ABB RAPID module: Module1.mod

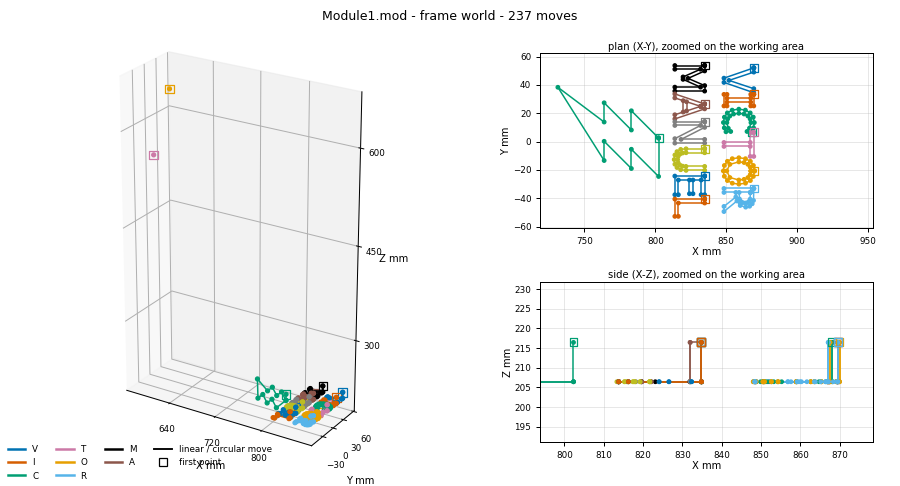
[picture p0: tool path of Module1.mod in frame world, 237 of 237 moves have a stored position in this frame; points joined in program order, loops and branches not executed]
MODULE Module1
        CONST robtarget Target_10_2:=[[151.956,135.501,-10],[0.707106781,0,0,0.707106781],[0,-2,1,0],[9E+09,9E+09,9E+09,9E+09,9E+09,9E+09]];
    CONST robtarget Target_10:=[[151.956,135.501,0],[0.707106781,0,0,0.707106781],[0,0,0,0],[9E+09,9E+09,9E+09,9E+09,9E+09,9E+09]];
    CONST robtarget Target_20:=[[154.96,135.501,0],[0.707106781,0,0,0.707106781],[0,-2,1,0],[9E+09,9E+09,9E+09,9E+09,9E+09,9E+09]];
    CONST robtarget Target_30:=[[160.796,152.992,0],[0.707106781,0,0,0.707106781],[0,-2,1,0],[9E+09,9E+09,9E+09,9E+09,9E+09,9E+09]];
    CONST robtarget Target_40:=[[166.632,135.501,0],[0.707106781,0,0,0.707106781],[0,-2,1,0],[9E+09,9E+09,9E+09,9E+09,9E+09,9E+09]];
    CONST robtarget Target_50:=[[169.481,135.501,0],[0.707106781,0,0,0.707106781],[0,-2,1,0],[9E+09,9E+09,9E+09,9E+09,9E+09,9E+09]];
    CONST robtarget Target_60:=[[162.229,156.559,0],[0.707106781,0,0,0.707106781],[0,-2,1,0],[9E+09,9E+09,9E+09,9E+09,9E+09,9E+09]];
    CONST robtarget Target_70:=[[159.209,156.559,0],[0.707106781,0,0,0.707106781],[0,-2,1,0],[9E+09,9E+09,9E+09,9E+09,9E+09,9E+09]];
    CONST robtarget Target_80:=[[151.956,135.501,0],[0.707106781,0,0,0.707106781],[0,-2,1,0],[9E+09,9E+09,9E+09,9E+09,9E+09,9E+09]];
    CONST robtarget Target_90_2:=[[170.676,135.501,-10],[0.707106781,0,0,0.707106781],[0,-2,1,0],[9E+09,9E+09,9E+09,9E+09,9E+09,9E+09]];
    CONST robtarget Target_90:=[[170.676,135.501,0],[0.707106781,0,0,0.707106781],[0,-2,1,0],[9E+09,9E+09,9E+09,9E+09,9E+09,9E+09]];
    CONST robtarget Target_100:=[[178.833,135.501,0],[0.707106781,0,0,0.707106781],[0,-2,1,0],[9E+09,9E+09,9E+09,9E+09,9E+09,9E+09]];
    CONST robtarget Target_110:=[[178.833,137.651,0],[0.707106781,0,0,0.707106781],[0,-2,1,0],[9E+09,9E+09,9E+09,9E+09,9E+09,9E+09]];
    CONST robtarget Target_120:=[[176.153,137.651,0],[0.707106781,0,0,0.707106781],[0,-2,1,0],[9E+09,9E+09,9E+09,9E+09,9E+09,9E+09]];
    CONST robtarget Target_130:=[[176.153,154.408,0],[0.707106781,0,0,0.707106781],[0,-2,1,0],[9E+09,9E+09,9E+09,9E+09,9E+09,9E+09]];
    CONST robtarget Target_140:=[[178.833,154.408,0],[0.707106781,0,0,0.707106781],[0,-2,1,0],[9E+09,9E+09,9E+09,9E+09,9E+09,9E+09]];
    CONST robtarget Target_150:=[[178.833,156.559,0],[0.707106781,0,0,0.707106781],[0,-2,1,0],[9E+09,9E+09,9E+09,9E+09,9E+09,9E+09]];
    CONST robtarget Target_160:=[[170.676,156.559,0],[0.707106781,0,0,0.707106781],[0,-2,1,0],[9E+09,9E+09,9E+09,9E+09,9E+09,9E+09]];
    CONST robtarget Target_170:=[[170.676,154.408,0],[0.707106781,0,0,0.707106781],[0,-2,1,0],[9E+09,9E+09,9E+09,9E+09,9E+09,9E+09]];
    CONST robtarget Target_180:=[[173.355,154.408,0],[0.707106781,0,0,0.707106781],[0,-2,1,0],[9E+09,9E+09,9E+09,9E+09,9E+09,9E+09]];
    CONST robtarget Target_190:=[[173.355,137.651,0],[0.707106781,0,0,0.707106781],[0,-2,1,0],[9E+09,9E+09,9E+09,9E+09,9E+09,9E+09]];
    CONST robtarget Target_200:=[[170.676,137.651,0],[0.707106781,0,0,0.707106781],[0,-2,1,0],[9E+09,9E+09,9E+09,9E+09,9E+09,9E+09]];
    CONST robtarget Target_210:=[[170.676,135.501,0],[0.707106781,0,0,0.707106781],[0,-2,1,0],[9E+09,9E+09,9E+09,9E+09,9E+09,9E+09]];
    CONST robtarget Target_220_2:=[[197.074,136.9,-10],[0.707106781,0,0,0.707106781],[0,-1,0,0],[9E+09,9E+09,9E+09,9E+09,9E+09,9E+09]];
    CONST robtarget Target_220:=[[197.074,136.9,0],[0.707106781,0,0,0.707106781],[0,0,0,0],[9E+09,9E+09,9E+09,9E+09,9E+09,9E+09]];
    CONST robtarget Target_230:=[[196.852,140.279,0],[0.707106781,0,0,0.707106781],[0,-1,0,0],[9E+09,9E+09,9E+09,9E+09,9E+09,9E+09]];
    CONST robtarget Target_240:=[[194.48,138.522,0],[0.707106781,0,0,0.707106781],[0,-1,0,0],[9E+09,9E+09,9E+09,9E+09,9E+09,9E+09]];
    CONST robtarget Target_250:=[[190.556,137.515,0],[0.707106781,0,0,0.707106781],[0,-1,0,0],[9E+09,9E+09,9E+09,9E+09,9E+09,9E+09]];
    CONST robtarget Target_260:=[[188.005,138.069,0],[0.707106781,0,0,0.707106781],[0,-1,0,0],[9E+09,9E+09,9E+09,9E+09,9E+09,9E+09]];
    CONST robtarget Target_270:=[[185.897,139.682,0],[0.707106781,0,0,0.707106781],[0,-1,0,0],[9E+09,9E+09,9E+09,9E+09,9E+09,9E+09]];
    CONST robtarget Target_280:=[[184.515,142.387,0],[0.707106781,0,0,0.707106781],[0,-1,0,0],[9E+09,9E+09,9E+09,9E+09,9E+09,9E+09]];
    CONST robtarget Target_290:=[[184.02,146.047,0],[0.707106781,0,0,0.707106781],[0,-1,0,0],[9E+09,9E+09,9E+09,9E+09,9E+09,9E+09]];
    CONST robtarget Target_300:=[[184.541,149.775,0],[0.707106781,0,0,0.707106781],[0,-2,1,0],[9E+09,9E+09,9E+09,9E+09,9E+09,9E+09]];
    CONST robtarget Target_310:=[[185.965,152.412,0],[0.707106781,0,0,0.707106781],[0,-2,1,0],[9E+09,9E+09,9E+09,9E+09,9E+09,9E+09]];
    CONST robtarget Target_320:=[[188.039,153.982,0],[0.707106781,0,0,0.707106781],[0,-2,1,0],[9E+09,9E+09,9E+09,9E+09,9E+09,9E+09]];
    CONST robtarget Target_330:=[[190.556,154.511,0],[0.707106781,0,0,0.707106781],[0,-2,1,0],[9E+09,9E+09,9E+09,9E+09,9E+09,9E+09]];
    CONST robtarget Target_340:=[[194.634,153.47,0],[0.707106781,0,0,0.707106781],[0,-2,1,0],[9E+09,9E+09,9E+09,9E+09,9E+09,9E+09]];
    CONST robtarget Target_350:=[[196.869,151.781,0],[0.707106781,0,0,0.707106781],[0,-2,1,0],[9E+09,9E+09,9E+09,9E+09,9E+09,9E+09]];
    CONST robtarget Target_360:=[[197.074,155.125,0],[0.707106781,0,0,0.707106781],[0,-2,1,0],[9E+09,9E+09,9E+09,9E+09,9E+09,9E+09]];
    CONST robtarget Target_370:=[[194.276,156.32,0],[0.707106781,0,0,0.707106781],[0,-2,1,0],[9E+09,9E+09,9E+09,9E+09,9E+09,9E+09]];
    CONST robtarget Target_380:=[[190.522,156.934,0],[0.707106781,0,0,0.707106781],[0,-2,1,0],[9E+09,9E+09,9E+09,9E+09,9E+09,9E+09]];
    CONST robtarget Target_390:=[[186.742,156.243,0],[0.707106781,0,0,0.707106781],[0,-2,1,0],[9E+09,9E+09,9E+09,9E+09,9E+09,9E+09]];
    CONST robtarget Target_400:=[[183.747,154.17,0],[0.707106781,0,0,0.707106781],[0,-2,1,0],[9E+09,9E+09,9E+09,9E+09,9E+09,9E+09]];
    CONST robtarget Target_410:=[[181.793,150.757,0],[0.707106781,0,0,0.707106781],[0,-2,1,0],[9E+09,9E+09,9E+09,9E+09,9E+09,9E+09]];
    CONST robtarget Target_420:=[[181.102,146.047,0],[0.707106781,0,0,0.707106781],[0,-1,0,0],[9E+09,9E+09,9E+09,9E+09,9E+09,9E+09]];
    CONST robtarget Target_430:=[[181.776,141.44,0],[0.707106781,0,0,0.707106781],[0,0,0,0],[9E+09,9E+09,9E+09,9E+09,9E+09,9E+09]];
    CONST robtarget Target_440:=[[183.73,138.027,0],[0.707106781,0,0,0.707106781],[0,0,0,0],[9E+09,9E+09,9E+09,9E+09,9E+09,9E+09]];
    CONST robtarget Target_450:=[[186.716,135.868,0],[0.707106781,0,0,0.707106781],[0,0,0,0],[9E+09,9E+09,9E+09,9E+09,9E+09,9E+09]];
    CONST robtarget Target_460:=[[190.573,135.126,0],[0.707106781,0,0,0.707106781],[0,0,0,0],[9E+09,9E+09,9E+09,9E+09,9E+09,9E+09]];
    CONST robtarget Target_470:=[[194.276,135.672,0],[0.707106781,0,0,0.707106781],[0,0,0,0],[9E+09,9E+09,9E+09,9E+09,9E+09,9E+09]];
    CONST robtarget Target_480:=[[197.074,136.9,0],[0.707106781,0,0,0.707106781],[0,0,0,0],[9E+09,9E+09,9E+09,9E+09,9E+09,9E+09]];
    CONST robtarget Target_490_2:=[[197.535,135.501,-10],[0.707106781,0,0,0.707106781],[0,-1,0,0],[9E+09,9E+09,9E+09,9E+09,9E+09,9E+09]];
    CONST robtarget Target_490:=[[197.535,135.501,0],[0.707106781,0,0,0.707106781],[0,0,0,0],[9E+09,9E+09,9E+09,9E+09,9E+09,9E+09]];
    CONST robtarget Target_500:=[[214.463,135.501,0],[0.707106781,0,0,0.707106781],[-1,0,-1,0],[9E+09,9E+09,9E+09,9E+09,9E+09,9E+09]];
    CONST robtarget Target_510:=[[214.463,137.993,0],[0.707106781,0,0,0.707106781],[-1,0,-1,0],[9E+09,9E+09,9E+09,9E+09,9E+09,9E+09]];
    CONST robtarget Target_520:=[[207.398,137.993,0],[0.707106781,0,0,0.707106781],[-1,0,-1,0],[9E+09,9E+09,9E+09,9E+09,9E+09,9E+09]];
    CONST robtarget Target_530:=[[207.398,156.559,0],[0.707106781,0,0,0.707106781],[-1,1,-2,0],[9E+09,9E+09,9E+09,9E+09,9E+09,9E+09]];
    CONST robtarget Target_540:=[[204.6,156.559,0],[0.707106781,0,0,0.707106781],[-1,1,-2,0],[9E+09,9E+09,9E+09,9E+09,9E+09,9E+09]];
    CONST robtarget Target_550:=[[204.6,137.993,0],[0.707106781,0,0,0.707106781],[-1,0,-1,0],[9E+09,9E+09,9E+09,9E+09,9E+09,9E+09]];
    CONST robtarget Target_560:=[[197.535,137.993,0],[0.707106781,0,0,0.707106781],[0,-1,0,0],[9E+09,9E+09,9E+09,9E+09,9E+09,9E+09]];
    CONST robtarget Target_570:=[[197.535,135.501,0],[0.707106781,0,0,0.707106781],[0,-1,0,0],[9E+09,9E+09,9E+09,9E+09,9E+09,9E+09]];
    CONST robtarget Target_580_2:=[[224.701,135.058,-10],[0.707106781,0,0,0.707106781],[-1,0,-1,0],[9E+09,9E+09,9E+09,9E+09,9E+09,9E+09]];
    CONST robtarget Target_580:=[[224.701,135.058,0],[0.707106781,0,0,0.707106781],[0,0,0,0],[9E+09,9E+09,9E+09,9E+09,9E+09,9E+09]];
    CONST robtarget Target_590:=[[228.575,135.808,0],[0.707106781,0,0,0.707106781],[-1,0,-1,0],[9E+09,9E+09,9E+09,9E+09,9E+09,9E+09]];
    CONST robtarget Target_600:=[[231.493,137.907,0],[0.707106781,0,0,0.707106781],[-1,0,-1,0],[9E+09,9E+09,9E+09,9E+09,9E+09,9E+09]];
    CONST robtarget Target_610:=[[233.353,141.354,0],[0.707106781,0,0,0.707106781],[-1,0,-1,0],[9E+09,9E+09,9E+09,9E+09,9E+09,9E+09]];
    CONST robtarget Target_620:=[[234.018,146.03,0],[0.707106781,0,0,0.707106781],[-1,0,-1,0],[9E+09,9E+09,9E+09,9E+09,9E+09,9E+09]];
    CONST robtarget Target_630:=[[233.37,150.663,0],[0.707106781,0,0,0.707106781],[-1,0,-1,0],[9E+09,9E+09,9E+09,9E+09,9E+09,9E+09]];
    CONST robtarget Target_640:=[[231.493,154.135,0],[0.707106781,0,0,0.707106781],[-1,0,-1,0],[9E+09,9E+09,9E+09,9E+09,9E+09,9E+09]];
    CONST robtarget Target_650:=[[228.481,156.303,0],[0.707106781,0,0,0.707106781],[-1,0,-1,0],[9E+09,9E+09,9E+09,9E+09,9E+09,9E+09]];
    CONST robtarget Target_660:=[[224.701,157.002,0],[0.707106781,0,0,0.707106781],[-1,0,-1,0],[9E+09,9E+09,9E+09,9E+09,9E+09,9E+09]];
    CONST robtarget Target_670:=[[220.862,156.277,0],[0.707106781,0,0,0.707106781],[-1,0,-1,0],[9E+09,9E+09,9E+09,9E+09,9E+09,9E+09]];
    CONST robtarget Target_680:=[[217.91,154.135,0],[0.707106781,0,0,0.707106781],[-1,0,-1,0],[9E+09,9E+09,9E+09,9E+09,9E+09,9E+09]];
    CONST robtarget Target_690:=[[216.05,150.68,0],[0.707106781,0,0,0.707106781],[-1,0,-1,0],[9E+09,9E+09,9E+09,9E+09,9E+09,9E+09]];
    CONST robtarget Target_700:=[[215.401,146.03,0],[0.707106781,0,0,0.707106781],[-1,0,-1,0],[9E+09,9E+09,9E+09,9E+09,9E+09,9E+09]];
    CONST robtarget Target_710:=[[216.058,141.371,0],[0.707106781,0,0,0.707106781],[-1,0,-1,0],[9E+09,9E+09,9E+09,9E+09,9E+09,9E+09]];
    CONST robtarget Target_720:=[[217.927,137.907,0],[0.707106781,0,0,0.707106781],[-1,0,-1,0],[9E+09,9E+09,9E+09,9E+09,9E+09,9E+09]];
    CONST robtarget Target_730:=[[220.87,135.783,0],[0.707106781,0,0,0.707106781],[-1,0,-1,0],[9E+09,9E+09,9E+09,9E+09,9E+09,9E+09]];
    CONST robtarget Target_740:=[[224.701,135.058,0],[0.707106781,0,0,0.707106781],[-1,0,-1,0],[9E+09,9E+09,9E+09,9E+09,9E+09,9E+09]];
    CONST robtarget Target_750_2:=[[224.718,137.481,-10],[0.707106781,0,0,0.707106781],[-1,0,-1,0],[9E+09,9E+09,9E+09,9E+09,9E+09,9E+09]];
    CONST robtarget Target_750:=[[224.718,137.481,0],[0.707106781,0,0,0.707106781],[-1,0,-1,0],[9E+09,9E+09,9E+09,9E+09,9E+09,9E+09]];
    CONST robtarget Target_760:=[[227.363,138.027,0],[0.707106781,0,0,0.707106781],[-1,0,-1,0],[9E+09,9E+09,9E+09,9E+09,9E+09,9E+09]];
    CONST robtarget Target_770:=[[229.377,139.665,0],[0.707106781,0,0,0.707106781],[-1,0,-1,0],[9E+09,9E+09,9E+09,9E+09,9E+09,9E+09]];
    CONST robtarget Target_780:=[[230.648,142.335,0],[0.707106781,0,0,0.707106781],[-1,0,-1,0],[9E+09,9E+09,9E+09,9E+09,9E+09,9E+09]];
    CONST robtarget Target_790:=[[231.1,146.03,0],[0.707106781,0,0,0.707106781],[-1,0,-1,0],[9E+09,9E+09,9E+09,9E+09,9E+09,9E+09]];
    CONST robtarget Target_800:=[[229.368,152.378,0],[0.707106781,0,0,0.707106781],[-1,0,-1,0],[9E+09,9E+09,9E+09,9E+09,9E+09,9E+09]];
    CONST robtarget Target_810:=[[224.718,154.579,0],[0.707106781,0,0,0.707106781],[-1,0,-1,0],[9E+09,9E+09,9E+09,9E+09,9E+09,9E+09]];
    CONST robtarget Target_820:=[[220.06,152.378,0],[0.707106781,0,0,0.707106781],[-1,0,-1,0],[9E+09,9E+09,9E+09,9E+09,9E+09,9E+09]];
    CONST robtarget Target_830:=[[218.319,146.03,0],[0.707106781,0,0,0.707106781],[-1,0,-1,0],[9E+09,9E+09,9E+09,9E+09,9E+09,9E+09]];
    CONST robtarget Target_840:=[[218.763,142.361,0],[0.707106781,0,0,0.707106781],[-1,0,-1,0],[9E+09,9E+09,9E+09,9E+09,9E+09,9E+09]];
    CONST robtarget Target_850:=[[220.043,139.665,0],[0.707106781,0,0,0.707106781],[-1,0,-1,0],[9E+09,9E+09,9E+09,9E+09,9E+09,9E+09]];
    CONST robtarget Target_860:=[[222.056,138.01,0],[0.707106781,0,0,0.707106781],[-1,0,-1,0],[9E+09,9E+09,9E+09,9E+09,9E+09,9E+09]];
    CONST robtarget Target_870:=[[224.718,137.481,0],[0.707106781,0,0,0.707106781],[-1,0,-1,0],[9E+09,9E+09,9E+09,9E+09,9E+09,9E+09]];
    CONST robtarget Target_880_2:=[[237.09,135.501,-10],[0.707106781,0,0,0.707106781],[-1,0,-1,0],[9E+09,9E+09,9E+09,9E+09,9E+09,9E+09]];
    CONST robtarget Target_880:=[[237.09,135.501,0],[0.707106781,0,0,0.707106781],[0,0,0,0],[9E+09,9E+09,9E+09,9E+09,9E+09,9E+09]];
    CONST robtarget Target_890:=[[245.545,135.697,0],[0.707106781,0,0,0.707106781],[-1,0,-1,0],[9E+09,9E+09,9E+09,9E+09,9E+09,9E+09]];
    CONST robtarget Target_900:=[[247.875,136.61,0],[0.707106781,0,0,0.707106781],[-1,0,-1,0],[9E+09,9E+09,9E+09,9E+09,9E+09,9E+09]];
    CONST robtarget Target_910:=[[249.624,138.445,0],[0.707106781,0,0,0.707106781],[-1,0,-1,0],[9E+09,9E+09,9E+09,9E+09,9E+09,9E+09]];
    CONST robtarget Target_920:=[[250.264,141.218,0],[0.707106781,0,0,0.707106781],[-1,0,-1,0],[9E+09,9E+09,9E+09,9E+09,9E+09,9E+09]];
    CONST robtarget Target_930:=[[249.086,145.083,0],[0.707106781,0,0,0.707106781],[-1,0,-1,0],[9E+09,9E+09,9E+09,9E+09,9E+09,9E+09]];
    CONST robtarget Target_940:=[[245.895,147.395,0],[0.707106781,0,0,0.707106781],[-1,0,-1,0],[9E+09,9E+09,9E+09,9E+09,9E+09,9E+09]];
    CONST robtarget Target_950:=[[253.386,156.559,0],[0.707106781,0,0,0.707106781],[-1,0,-1,0],[9E+09,9E+09,9E+09,9E+09,9E+09,9E+09]];
    CONST robtarget Target_960:=[[249.752,156.559,0],[0.707106781,0,0,0.707106781],[-1,0,-1,0],[9E+09,9E+09,9E+09,9E+09,9E+09,9E+09]];
    CONST robtarget Target_970:=[[243.097,148.18,0],[0.707106781,0,0,0.707106781],[-1,0,-1,0],[9E+09,9E+09,9E+09,9E+09,9E+09,9E+09]];
    CONST robtarget Target_980:=[[239.889,148.18,0],[0.707106781,0,0,0.707106781],[-1,0,-1,0],[9E+09,9E+09,9E+09,9E+09,9E+09,9E+09]];
    CONST robtarget Target_990:=[[239.889,156.559,0],[0.707106781,0,0,0.707106781],[-1,0,-1,0],[9E+09,9E+09,9E+09,9E+09,9E+09,9E+09]];
    CONST robtarget Target_1000:=[[237.09,156.559,0],[0.707106781,0,0,0.707106781],[-1,0,-1,0],[9E+09,9E+09,9E+09,9E+09,9E+09,9E+09]];
    CONST robtarget Target_1010:=[[237.09,135.501,0],[0.707106781,0,0,0.707106781],[0,0,0,0],[9E+09,9E+09,9E+09,9E+09,9E+09,9E+09]];
    CONST robtarget Target_1020_2:=[[239.889,137.924,-10],[0.707106781,0,0,0.707106781],[0,0,0,0],[9E+09,9E+09,9E+09,9E+09,9E+09,9E+09]];
    CONST robtarget Target_1020:=[[239.889,137.924,0],[0.707106781,0,0,0.707106781],[0,0,0,0],[9E+09,9E+09,9E+09,9E+09,9E+09,9E+09]];
    CONST robtarget Target_1030:=[[244.624,138.086,0],[0.707106781,0,0,0.707106781],[0,0,0,0],[9E+09,9E+09,9E+09,9E+09,9E+09,9E+09]];
    CONST robtarget Target_1040:=[[246.015,138.641,0],[0.707106781,0,0,0.707106781],[0,0,0,0],[9E+09,9E+09,9E+09,9E+09,9E+09,9E+09]];
    CONST robtarget Target_1050:=[[247.021,139.81,0],[0.707106781,0,0,0.707106781],[0,0,0,0],[9E+09,9E+09,9E+09,9E+09,9E+09,9E+09]];
    CONST robtarget Target_1060:=[[247.346,141.44,0],[0.707106781,0,0,0.707106781],[0,0,0,0],[9E+09,9E+09,9E+09,9E+09,9E+09,9E+09]];
    CONST robtarget Target_1070:=[[247.056,143.351,0],[0.707106781,0,0,0.707106781],[0,0,0,0],[9E+09,9E+09,9E+09,9E+09,9E+09,9E+09]];
    CONST robtarget Target_1080:=[[246.151,144.75,0],[0.707106781,0,0,0.707106781],[0,0,0,0],[9E+09,9E+09,9E+09,9E+09,9E+09,9E+09]];
    CONST robtarget Target_1090:=[[244.522,145.629,0],[0.707106781,0,0,0.707106781],[0,0,0,0],[9E+09,9E+09,9E+09,9E+09,9E+09,9E+09]];
    CONST robtarget Target_1100:=[[239.889,145.842,0],[0.707106781,0,0,0.707106781],[0,0,0,0],[9E+09,9E+09,9E+09,9E+09,9E+09,9E+09]];
    CONST robtarget Target_1110:=[[239.889,137.924,0],[0.707106781,0,0,0.707106781],[0,0,0,0],[9E+09,9E+09,9E+09,9E+09,9E+09,9E+09]];
    CONST robtarget Target_1120_2:=[[150.301,170.172,-10],[0.707106781,0,0,0.707106781],[0,-1,0,0],[9E+09,9E+09,9E+09,9E+09,9E+09,9E+09]];
    CONST robtarget Target_1120:=[[150.301,170.172,0],[0.707106781,0,0,0.707106781],[0,0,0,0],[9E+09,9E+09,9E+09,9E+09,9E+09,9E+09]];
    CONST robtarget Target_1130:=[[154.123,170.172,0],[0.707106781,0,0,0.707106781],[0,-1,0,0],[9E+09,9E+09,9E+09,9E+09,9E+09,9E+09]];
    CONST robtarget Target_1140:=[[159.379,181.895,0],[0.707106781,0,0,0.707106781],[0,-1,0,0],[9E+09,9E+09,9E+09,9E+09,9E+09,9E+09]];
    CONST robtarget Target_1150:=[[164.464,170.172,0],[0.707106781,0,0,0.707106781],[0,-1,0,0],[9E+09,9E+09,9E+09,9E+09,9E+09,9E+09]];
    CONST robtarget Target_1160:=[[168.355,170.172,0],[0.707106781,0,0,0.707106781],[0,-1,0,0],[9E+09,9E+09,9E+09,9E+09,9E+09,9E+09]];
    CONST robtarget Target_1170:=[[168.355,191.229,0],[0.707106781,0,0,0.707106781],[0,-1,0,0],[9E+09,9E+09,9E+09,9E+09,9E+09,9E+09]];
    CONST robtarget Target_1180:=[[165.557,191.229,0],[0.707106781,0,0,0.707106781],[0,-1,0,0],[9E+09,9E+09,9E+09,9E+09,9E+09,9E+09]];
    CONST robtarget Target_1190:=[[165.557,173.09,0],[0.707106781,0,0,0.707106781],[0,-1,0,0],[9E+09,9E+09,9E+09,9E+09,9E+09,9E+09]];
    CONST robtarget Target_1200:=[[160.062,185.427,0],[0.707106781,0,0,0.707106781],[0,-1,0,0],[9E+09,9E+09,9E+09,9E+09,9E+09,9E+09]];
    CONST robtarget Target_1210:=[[158.355,185.427,0],[0.707106781,0,0,0.707106781],[0,-1,0,0],[9E+09,9E+09,9E+09,9E+09,9E+09,9E+09]];
    CONST robtarget Target_1220:=[[152.912,173.09,0],[0.707106781,0,0,0.707106781],[0,-1,0,0],[9E+09,9E+09,9E+09,9E+09,9E+09,9E+09]];
    CONST robtarget Target_1230:=[[152.912,191.229,0],[0.707106781,0,0,0.707106781],[0,-1,0,0],[9E+09,9E+09,9E+09,9E+09,9E+09,9E+09]];
    CONST robtarget Target_1240:=[[150.301,191.229,0],[0.707106781,0,0,0.707106781],[0,-1,0,0],[9E+09,9E+09,9E+09,9E+09,9E+09,9E+09]];
    CONST robtarget Target_1250:=[[150.301,170.172,0],[0.707106781,0,0,0.707106781],[0,-1,0,0],[9E+09,9E+09,9E+09,9E+09,9E+09,9E+09]];
    CONST robtarget Target_1260_2:=[[177.45,170.172,-10],[0.707106781,0,0,0.707106781],[0,-1,0,0],[9E+09,9E+09,9E+09,9E+09,9E+09,9E+09]];
    CONST robtarget Target_1260:=[[177.45,170.172,0],[0.707106781,0,0,0.707106781],[0,0,0,0],[9E+09,9E+09,9E+09,9E+09,9E+09,9E+09]];
    CONST robtarget Target_1270:=[[180.897,170.172,0],[0.707106781,0,0,0.707106781],[0,-1,0,0],[9E+09,9E+09,9E+09,9E+09,9E+09,9E+09]];
    CONST robtarget Target_1280:=[[187.996,191.229,0],[0.707106781,0,0,0.707106781],[0,-1,0,0],[9E+09,9E+09,9E+09,9E+09,9E+09,9E+09]];
    CONST robtarget Target_1290:=[[185.044,191.229,0],[0.707106781,0,0,0.707106781],[0,-1,0,0],[9E+09,9E+09,9E+09,9E+09,9E+09,9E+09]];
    CONST robtarget Target_1300:=[[183.133,185.342,0],[0.707106781,0,0,0.707106781],[0,-1,0,0],[9E+09,9E+09,9E+09,9E+09,9E+09,9E+09]];
    CONST robtarget Target_1310:=[[175.095,185.342,0],[0.707106781,0,0,0.707106781],[0,-1,0,0],[9E+09,9E+09,9E+09,9E+09,9E+09,9E+09]];
    CONST robtarget Target_1320:=[[173.184,191.229,0],[0.707106781,0,0,0.707106781],[0,-1,0,0],[9E+09,9E+09,9E+09,9E+09,9E+09,9E+09]];
    CONST robtarget Target_1330:=[[170.352,191.229,0],[0.707106781,0,0,0.707106781],[0,-1,0,0],[9E+09,9E+09,9E+09,9E+09,9E+09,9E+09]];
    CONST robtarget Target_1340:=[[177.45,170.172,0],[0.707106781,0,0,0.707106781],[0,-1,0,0],[9E+09,9E+09,9E+09,9E+09,9E+09,9E+09]];
    CONST robtarget Target_1350_2:=[[179.106,173.038,-10],[0.707106781,0,0,0.707106781],[0,-1,0,0],[9E+09,9E+09,9E+09,9E+09,9E+09,9E+09]];
    CONST robtarget Target_1350:=[[179.106,173.038,0],[0.707106781,0,0,0.707106781],[0,-1,0,0],[9E+09,9E+09,9E+09,9E+09,9E+09,9E+09]];
    CONST robtarget Target_1360:=[[182.365,182.953,0],[0.707106781,0,0,0.707106781],[0,-1,0,0],[9E+09,9E+09,9E+09,9E+09,9E+09,9E+09]];
    CONST robtarget Target_1370:=[[175.863,182.953,0],[0.707106781,0,0,0.707106781],[0,-1,0,0],[9E+09,9E+09,9E+09,9E+09,9E+09,9E+09]];
    CONST robtarget Target_1380:=[[179.106,173.038,0],[0.707106781,0,0,0.707106781],[0,-1,0,0],[9E+09,9E+09,9E+09,9E+09,9E+09,9E+09]];
    CONST robtarget Target_1390_2:=[[189.993,170.172,-10],[0.707106781,0,0,0.707106781],[0,0,0,0],[9E+09,9E+09,9E+09,9E+09,9E+09,9E+09]];
    CONST robtarget Target_1390:=[[189.993,170.172,0],[0.707106781,0,0,0.707106781],[0,0,0,0],[9E+09,9E+09,9E+09,9E+09,9E+09,9E+09]];
    CONST robtarget Target_1400:=[[193.969,170.172,0],[0.707106781,0,0,0.707106781],[0,0,0,0],[9E+09,9E+09,9E+09,9E+09,9E+09,9E+09]];
    CONST robtarget Target_1410:=[[202.45,186.843,0],[0.707106781,0,0,0.707106781],[0,0,0,0],[9E+09,9E+09,9E+09,9E+09,9E+09,9E+09]];
    CONST robtarget Target_1420:=[[202.45,170.172,0],[0.707106781,0,0,0.707106781],[0,0,0,0],[9E+09,9E+09,9E+09,9E+09,9E+09,9E+09]];
    CONST robtarget Target_1430:=[[205.06,170.172,0],[0.707106781,0,0,0.707106781],[0,0,0,0],[9E+09,9E+09,9E+09,9E+09,9E+09,9E+09]];
    CONST robtarget Target_1440:=[[205.06,191.229,0],[0.707106781,0,0,0.707106781],[0,0,0,0],[9E+09,9E+09,9E+09,9E+09,9E+09,9E+09]];
    CONST robtarget Target_1450:=[[201.921,191.229,0],[0.707106781,0,0,0.707106781],[0,0,0,0],[9E+09,9E+09,9E+09,9E+09,9E+09,9E+09]];
    CONST robtarget Target_1460:=[[192.603,173.072,0],[0.707106781,0,0,0.707106781],[0,0,0,0],[9E+09,9E+09,9E+09,9E+09,9E+09,9E+09]];
    CONST robtarget Target_1470:=[[192.603,191.229,0],[0.707106781,0,0,0.707106781],[0,0,0,0],[9E+09,9E+09,9E+09,9E+09,9E+09,9E+09]];
    CONST robtarget Target_1480:=[[189.993,191.229,0],[0.707106781,0,0,0.707106781],[0,0,0,0],[9E+09,9E+09,9E+09,9E+09,9E+09,9E+09]];
    CONST robtarget Target_1490:=[[189.993,170.172,0],[0.707106781,0,0,0.707106781],[0,0,0,0],[9E+09,9E+09,9E+09,9E+09,9E+09,9E+09]];
    CONST robtarget Target_1500_2:=[[209.07,170.172,-10],[0.707106781,0,0,0.707106781],[-1,0,-1,0],[9E+09,9E+09,9E+09,9E+09,9E+09,9E+09]];
    CONST robtarget Target_1500:=[[209.07,170.172,0],[0.707106781,0,0,0.707106781],[0,0,0,0],[9E+09,9E+09,9E+09,9E+09,9E+09,9E+09]];
    CONST robtarget Target_1510:=[[211.869,170.172,0],[0.707106781,0,0,0.707106781],[0,0,0,0],[9E+09,9E+09,9E+09,9E+09,9E+09,9E+09]];
    CONST robtarget Target_1520:=[[211.869,183.311,0],[0.707106781,0,0,0.707106781],[0,0,0,0],[9E+09,9E+09,9E+09,9E+09,9E+09,9E+09]];
    CONST robtarget Target_1530:=[[212.057,185.768,0],[0.707106781,0,0,0.707106781],[0,0,0,0],[9E+09,9E+09,9E+09,9E+09,9E+09,9E+09]];
    CONST robtarget Target_1540:=[[212.773,187.56,0],[0.707106781,0,0,0.707106781],[0,0,0,0],[9E+09,9E+09,9E+09,9E+09,9E+09,9E+09]];
    CONST robtarget Target_1550:=[[214.309,188.848,0],[0.707106781,0,0,0.707106781],[0,0,0,0],[9E+09,9E+09,9E+09,9E+09,9E+09,9E+09]];
    CONST robtarget Target_1560:=[[216.681,189.284,0],[0.707106781,0,0,0.707106781],[0,0,0,0],[9E+09,9E+09,9E+09,9E+09,9E+09,9E+09]];
    CONST robtarget Target_1570:=[[219.019,188.848,0],[0.707106781,0,0,0.707106781],[0,0,0,0],[9E+09,9E+09,9E+09,9E+09,9E+09,9E+09]];
    CONST robtarget Target_1580:=[[220.606,187.56,0],[0.707106781,0,0,0.707106781],[0,0,0,0],[9E+09,9E+09,9E+09,9E+09,9E+09,9E+09]];
    CONST robtarget Target_1590:=[[221.323,185.777,0],[0.707106781,0,0,0.707106781],[0,0,0,0],[9E+09,9E+09,9E+09,9E+09,9E+09,9E+09]];
    CONST robtarget Target_1600:=[[221.51,183.379,0],[0.707106781,0,0,0.707106781],[0,0,0,0],[9E+09,9E+09,9E+09,9E+09,9E+09,9E+09]];
    CONST robtarget Target_1610:=[[221.51,170.172,0],[0.707106781,0,0,0.707106781],[0,0,0,0],[9E+09,9E+09,9E+09,9E+09,9E+09,9E+09]];
    CONST robtarget Target_1620:=[[224.309,170.172,0],[0.707106781,0,0,0.707106781],[0,0,0,0],[9E+09,9E+09,9E+09,9E+09,9E+09,9E+09]];
    CONST robtarget Target_1630:=[[224.309,183.311,0],[0.707106781,0,0,0.707106781],[0,0,0,0],[9E+09,9E+09,9E+09,9E+09,9E+09,9E+09]];
    CONST robtarget Target_1640:=[[223.865,187.082,0],[0.707106781,0,0,0.707106781],[0,0,0,0],[9E+09,9E+09,9E+09,9E+09,9E+09,9E+09]];
    CONST robtarget Target_1650:=[[222.295,189.727,0],[0.707106781,0,0,0.707106781],[0,0,0,0],[9E+09,9E+09,9E+09,9E+09,9E+09,9E+09]];
    CONST robtarget Target_1660:=[[219.957,191.195,0],[0.707106781,0,0,0.707106781],[0,0,0,0],[9E+09,9E+09,9E+09,9E+09,9E+09,9E+09]];
    CONST robtarget Target_1670:=[[216.681,191.673,0],[0.707106781,0,0,0.707106781],[0,0,0,0],[9E+09,9E+09,9E+09,9E+09,9E+09,9E+09]];
    CONST robtarget Target_1680:=[[213.439,191.186,0],[0.707106781,0,0,0.707106781],[0,0,0,0],[9E+09,9E+09,9E+09,9E+09,9E+09,9E+09]];
    CONST robtarget Target_1690:=[[211.084,189.727,0],[0.707106781,0,0,0.707106781],[0,0,0,0],[9E+09,9E+09,9E+09,9E+09,9E+09,9E+09]];
    CONST robtarget Target_1700:=[[209.523,187.099,0],[0.707106781,0,0,0.707106781],[0,0,0,0],[9E+09,9E+09,9E+09,9E+09,9E+09,9E+09]];
    CONST robtarget Target_1710:=[[209.07,183.311,0],[0.707106781,0,0,0.707106781],[0,0,0,0],[9E+09,9E+09,9E+09,9E+09,9E+09,9E+09]];
    CONST robtarget Target_1720:=[[209.07,170.172,0],[0.707106781,0,0,0.707106781],[0,0,0,0],[9E+09,9E+09,9E+09,9E+09,9E+09,9E+09]];
    CONST robtarget Target_1730_2:=[[228.319,170.172,-10],[0.707106781,0,0,0.707106781],[0,0,0,0],[9E+09,9E+09,9E+09,9E+09,9E+09,9E+09]];
    CONST robtarget Target_1730:=[[228.319,170.172,0],[0.707106781,0,0,0.707106781],[0,0,0,0],[9E+09,9E+09,9E+09,9E+09,9E+09,9E+09]];
    CONST robtarget Target_1740:=[[241.493,170.172,0],[0.707106781,0,0,0.707106781],[0,0,0,0],[9E+09,9E+09,9E+09,9E+09,9E+09,9E+09]];
    CONST robtarget Target_1750:=[[241.493,172.663,0],[0.707106781,0,0,0.707106781],[0,0,0,0],[9E+09,9E+09,9E+09,9E+09,9E+09,9E+09]];
    CONST robtarget Target_1760:=[[231.118,172.663,0],[0.707106781,0,0,0.707106781],[0,0,0,0],[9E+09,9E+09,9E+09,9E+09,9E+09,9E+09]];
    CONST robtarget Target_1770:=[[231.118,178.431,0],[0.707106781,0,0,0.707106781],[0,0,0,0],[9E+09,9E+09,9E+09,9E+09,9E+09,9E+09]];
    CONST robtarget Target_1780:=[[240.793,178.431,0],[0.707106781,0,0,0.707106781],[0,0,0,0],[9E+09,9E+09,9E+09,9E+09,9E+09,9E+09]];
    CONST robtarget Target_1790:=[[240.793,180.922,0],[0.707106781,0,0,0.707106781],[0,0,0,0],[9E+09,9E+09,9E+09,9E+09,9E+09,9E+09]];
    CONST robtarget Target_1800:=[[231.118,180.922,0],[0.707106781,0,0,0.707106781],[0,0,0,0],[9E+09,9E+09,9E+09,9E+09,9E+09,9E+09]];
    CONST robtarget Target_1810:=[[231.118,188.738,0],[0.707106781,0,0,0.707106781],[0,0,0,0],[9E+09,9E+09,9E+09,9E+09,9E+09,9E+09]];
    CONST robtarget Target_1820:=[[241.493,188.738,0],[0.707106781,0,0,0.707106781],[0,0,0,0],[9E+09,9E+09,9E+09,9E+09,9E+09,9E+09]];
    CONST robtarget Target_1830:=[[241.493,191.229,0],[0.707106781,0,0,0.707106781],[0,0,0,0],[9E+09,9E+09,9E+09,9E+09,9E+09,9E+09]];
    CONST robtarget Target_1840:=[[228.319,191.229,0],[0.707106781,0,0,0.707106781],[0,0,0,0],[9E+09,9E+09,9E+09,9E+09,9E+09,9E+09]];
    CONST robtarget Target_1850:=[[228.319,170.172,0],[0.707106781,0,0,0.707106781],[0,0,0,0],[9E+09,9E+09,9E+09,9E+09,9E+09,9E+09]];
    CONST robtarget Target_1860_2:=[[244.564,170.172,-10],[0.707106781,0,0,0.707106781],[0,0,0,0],[9E+09,9E+09,9E+09,9E+09,9E+09,9E+09]];
    CONST robtarget Target_1860:=[[244.564,170.172,0],[0.707106781,0,0,0.707106781],[0,0,0,0],[9E+09,9E+09,9E+09,9E+09,9E+09,9E+09]];
    CONST robtarget Target_1870:=[[247.363,170.172,0],[0.707106781,0,0,0.707106781],[0,0,0,0],[9E+09,9E+09,9E+09,9E+09,9E+09,9E+09]];
    CONST robtarget Target_1880:=[[247.363,188.738,0],[0.707106781,0,0,0.707106781],[0,0,0,0],[9E+09,9E+09,9E+09,9E+09,9E+09,9E+09]];
    CONST robtarget Target_1890:=[[256.765,188.738,0],[0.707106781,0,0,0.707106781],[0,0,0,0],[9E+09,9E+09,9E+09,9E+09,9E+09,9E+09]];
    CONST robtarget Target_1900:=[[256.765,191.229,0],[0.707106781,0,0,0.707106781],[0,0,0,0],[9E+09,9E+09,9E+09,9E+09,9E+09,9E+09]];
    CONST robtarget Target_1910:=[[244.564,191.229,0],[0.707106781,0,0,0.707106781],[0,0,0,0],[9E+09,9E+09,9E+09,9E+09,9E+09,9E+09]];
    CONST robtarget Target_1920:=[[244.564,170.172,0],[0.707106781,0,0,0.707106781],[0,0,0,0],[9E+09,9E+09,9E+09,9E+09,9E+09,9E+09]];
    CONST robtarget Target_1930_2:=[[201.446,202.7,-10],[0.707106781,0,0,0.707106781],[0,-2,1,0],[9E+09,9E+09,9E+09,9E+09,9E+09,9E+09]];
    CONST robtarget Target_1930:=[[201.446,202.7,0],[0.707106781,0,0,0.707106781],[0,0,0,0],[9E+09,9E+09,9E+09,9E+09,9E+09,9E+09]];
    CONST robtarget Target_1940:=[[228.616,202.7,0],[0.707106781,0,0,0.707106781],[0,0,0,0],[9E+09,9E+09,9E+09,9E+09,9E+09,9E+09]];
    CONST robtarget Target_1950:=[[209.404,221.912,0],[0.707106781,0,0,0.707106781],[0,0,0,0],[9E+09,9E+09,9E+09,9E+09,9E+09,9E+09]];
    CONST robtarget Target_1960:=[[222.989,221.912,0],[0.707106781,0,0,0.707106781],[0,0,0,0],[9E+09,9E+09,9E+09,9E+09,9E+09,9E+09]];
    CONST robtarget Target_1970:=[[203.777,241.124,0],[0.707106781,0,0,0.707106781],[0,0,0,0],[9E+09,9E+09,9E+09,9E+09,9E+09,9E+09]];
    CONST robtarget Target_1980:=[[217.362,241.124,0],[0.707106781,0,0,0.707106781],[0,0,0,0],[9E+09,9E+09,9E+09,9E+09,9E+09,9E+09]];
    CONST robtarget Target_1990:=[[165.644,273.791,0],[0.707106781,0,0,0.707106781],[0,0,0,0],[9E+09,9E+09,9E+09,9E+09,9E+09,9E+09]];
    CONST robtarget Target_2000:=[[190.192,241.124,0],[0.707106781,0,0,0.707106781],[0,0,0,0],[9E+09,9E+09,9E+09,9E+09,9E+09,9E+09]];
    CONST robtarget Target_2010:=[[176.607,241.124,0],[0.707106781,0,0,0.707106781],[0,0,0,0],[9E+09,9E+09,9E+09,9E+09,9E+09,9E+09]];
    CONST robtarget Target_2020:=[[195.819,221.912,0],[0.707106781,0,0,0.707106781],[0,0,0,0],[9E+09,9E+09,9E+09,9E+09,9E+09,9E+09]];
    CONST robtarget Target_2030:=[[182.234,221.912,0],[0.707106781,0,0,0.707106781],[0,0,0,0],[9E+09,9E+09,9E+09,9E+09,9E+09,9E+09]];
    CONST robtarget Target_2040:=[[201.446,202.7,0],[0.707106781,0,0,0.707106781],[0,0,0,0],[9E+09,9E+09,9E+09,9E+09,9E+09,9E+09]];
    CONST robtarget Target_2060_5:=[[109.64,110.982,0],[0.707106781,0,0,0.707106781],[0,0,0,0],[9E+09,9E+09,9E+09,9E+09,9E+09,9E+09]];
    CONST robtarget Target_2060:=[[109.64,110.982,0],[0.707106781,0,0,0.707106781],[0,0,0,0],[9E+09,9E+09,9E+09,9E+09,9E+09,9E+09]];
    CONST robtarget Target_2070:=[[109.64,290.982,0],[0.707106781,0,0,0.707106781],[0,0,0,0],[9E+09,9E+09,9E+09,9E+09,9E+09,9E+09]];
    CONST robtarget Target_2080:=[[289.64,290.982,0],[0.707106781,0,0,0.707106781],[0,0,0,0],[9E+09,9E+09,9E+09,9E+09,9E+09,9E+09]];
    CONST robtarget Target_2090:=[[289.64,110.982,0],[0.707106781,0,0,0.707106781],[0,0,0,0],[9E+09,9E+09,9E+09,9E+09,9E+09,9E+09]];
    PERS tooldata MyNewTool:=[TRUE,[[79.902999999,0,127.403],[0.923879533,0,0.382683431,0]],[0.1,[0,0,1],[1,0,0,0],0,0,0]];
    TASK PERS wobjdata Workobject_1:=[FALSE,TRUE,"",[[1005,204.006,206.452],[0,-0.707106781,0.707106781,0]],[[0,0,0],[1,0,0,0]]];
    CONST robtarget Target_2100:=[[204.006,428.326,-340.148],[0.707106781,0,0,0.707106781],[0,0,0,0],[9E+09,9E+09,9E+09,9E+09,9E+09,9E+09]];
    CONST robtarget Target_2110:=[[-429.595294319,508.357425752,-671.10646312],[0.612579887,0.241340938,-0.727509715,0.192950894],[0,-1,0,1],[9E+09,9E+09,9E+09,9E+09,9E+09,9E+09]];
    CONST robtarget Target_2120:=[[-23.442776222,446.747326228,-645.298589371],[0.228349534,0.861489909,0.443353827,-0.095545856],[0,-1,2,1],[9E+09,9E+09,9E+09,9E+09,9E+09,9E+09]];
    CONST robtarget Target_2130:=[[-213.64008263,445.141886894,-619.680858581],[0.68372228,0.288804128,-0.575754444,0.342961864],[0,0,-1,1],[9E+09,9E+09,9E+09,9E+09,9E+09,9E+09]];
    CONST robtarget Target_2140:=[[-117.115812609,437.380464058,-555.898830526],[0.654216666,0.328979684,-0.564091866,0.381540677],[0,0,-1,1],[9E+09,9E+09,9E+09,9E+09,9E+09,9E+09]];
    CONST robtarget Target_2150:=[[204.006,380.705938586,-619.675051892],[0.450873103,0.544714094,-0.544714094,0.450873103],[0,0,0,1],[9E+09,9E+09,9E+09,9E+09,9E+09,9E+09]];
    CONST robtarget Target_2160:=[[223.05767633,386.247950642,-455.700408414],[0.078798459,-0.437186278,-0.539494345,0.715265555],[-1,0,0,0],[9E+09,9E+09,9E+09,9E+09,9E+09,9E+09]];
!***********************************************************
    !
    ! Module:  Module1
    !
    ! Description:
    !   <Insert description here>
    !
    ! Author: macuser
    !
    ! Version: 1.0
    !
    !***********************************************************


    !***********************************************************
    !
    ! Procedure main
    !
    !   This is the entry point of your program
    !
    !***********************************************************
    PROC main()
        !Add your code here
        Reset DO_01;
        Reset DO_03;
        WHILE TRUE DO
            IF DI_01 = 1 THEN
                Set DO_01;
                HOME;
                V;
                I;
                C;
                T;
                O;
                R;
                M;
                A;
                N;
                U;
                E;
                L;
                RAYO;
                HOME;
                Reset DO_01;
            ENDIF
            IF DI_02 = 1 THEN
                Set DO_03;
                TC;
                Reset DO_03;
            ENDIF
        ENDWHILE

    ENDPROC
    PROC V()
        MoveL Target_10_2,v50,z100,MyNewTool\WObj:=Workobject_1;
        MoveL Target_10,v50,z100,MyNewTool\WObj:=Workobject_1;
        MoveL Target_20,v50,z100,MyNewTool\WObj:=Workobject_1;
        MoveL Target_30,v50,z100,MyNewTool\WObj:=Workobject_1;
        MoveL Target_40,v50,z100,MyNewTool\WObj:=Workobject_1;
        MoveL Target_50,v50,z100,MyNewTool\WObj:=Workobject_1;
        MoveL Target_60,v50,z100,MyNewTool\WObj:=Workobject_1;
        MoveL Target_70,v50,z100,MyNewTool\WObj:=Workobject_1;
        MoveL Target_80,v50,z100,MyNewTool\WObj:=Workobject_1;
        MoveL Target_10_2,v50,z100,MyNewTool\WObj:=Workobject_1;
    ENDPROC
    PROC I()
        MoveL Target_90_2,v50,z100,MyNewTool\WObj:=Workobject_1;
        MoveL Target_90,v50,z100,MyNewTool\WObj:=Workobject_1;
        MoveL Target_100,v50,z100,MyNewTool\WObj:=Workobject_1;
        MoveL Target_110,v50,z100,MyNewTool\WObj:=Workobject_1;
        MoveL Target_120,v50,z100,MyNewTool\WObj:=Workobject_1;
        MoveL Target_130,v50,z100,MyNewTool\WObj:=Workobject_1;
        MoveL Target_140,v50,z100,MyNewTool\WObj:=Workobject_1;
        MoveL Target_150,v50,z100,MyNewTool\WObj:=Workobject_1;
        MoveL Target_160,v50,z100,MyNewTool\WObj:=Workobject_1;
        MoveL Target_170,v50,z100,MyNewTool\WObj:=Workobject_1;
        MoveL Target_180,v50,z100,MyNewTool\WObj:=Workobject_1;
        MoveL Target_190,v50,z100,MyNewTool\WObj:=Workobject_1;
        MoveL Target_200,v50,z100,MyNewTool\WObj:=Workobject_1;
        MoveL Target_210,v50,z100,MyNewTool\WObj:=Workobject_1;
        MoveL Target_90_2,v50,z100,MyNewTool\WObj:=Workobject_1;
    ENDPROC
    PROC C()
        MoveL Target_220_2,v50,z0,MyNewTool\WObj:=Workobject_1;
        MoveL Target_220,v50,z0,MyNewTool\WObj:=Workobject_1;
        MoveL Target_230,v50,z0,MyNewTool\WObj:=Workobject_1;
        MoveL Target_240,v50,z0,MyNewTool\WObj:=Workobject_1;
        MoveL Target_250,v50,z0,MyNewTool\WObj:=Workobject_1;
        MoveL Target_260,v50,z0,MyNewTool\WObj:=Workobject_1;
        MoveL Target_270,v50,z0,MyNewTool\WObj:=Workobject_1;
        MoveL Target_280,v50,z0,MyNewTool\WObj:=Workobject_1;
        MoveL Target_290,v50,z0,MyNewTool\WObj:=Workobject_1;
        MoveL Target_300,v50,z0,MyNewTool\WObj:=Workobject_1;
        MoveL Target_310,v50,z0,MyNewTool\WObj:=Workobject_1;
        MoveL Target_320,v50,z0,MyNewTool\WObj:=Workobject_1;
        MoveL Target_330,v50,z0,MyNewTool\WObj:=Workobject_1;
        MoveL Target_340,v50,z0,MyNewTool\WObj:=Workobject_1;
        MoveL Target_350,v50,z0,MyNewTool\WObj:=Workobject_1;
        MoveL Target_360,v50,z0,MyNewTool\WObj:=Workobject_1;
        MoveL Target_370,v50,z0,MyNewTool\WObj:=Workobject_1;
        MoveL Target_380,v50,z0,MyNewTool\WObj:=Workobject_1;
        MoveL Target_390,v50,z0,MyNewTool\WObj:=Workobject_1;
        MoveL Target_400,v50,z0,MyNewTool\WObj:=Workobject_1;
        MoveL Target_410,v50,z0,MyNewTool\WObj:=Workobject_1;
        MoveL Target_420,v50,z0,MyNewTool\WObj:=Workobject_1;
        MoveL Target_430,v50,z0,MyNewTool\WObj:=Workobject_1;
        MoveL Target_440,v50,z0,MyNewTool\WObj:=Workobject_1;
        MoveL Target_450,v50,z0,MyNewTool\WObj:=Workobject_1;
        MoveL Target_460,v50,z0,MyNewTool\WObj:=Workobject_1;
        MoveL Target_470,v50,z0,MyNewTool\WObj:=Workobject_1;
        MoveL Target_480,v50,z0,MyNewTool\WObj:=Workobject_1;
        MoveL Target_220_2,v50,z0,MyNewTool\WObj:=Workobject_1;
    ENDPROC
    PROC T()
        MoveL Target_490_2,v50,z0,MyNewTool\WObj:=Workobject_1;
        MoveL Target_490,v50,z0,MyNewTool\WObj:=Workobject_1;
        MoveL Target_500,v50,z0,MyNewTool\WObj:=Workobject_1;
        MoveL Target_510,v50,z0,MyNewTool\WObj:=Workobject_1;
        MoveL Target_520,v50,z0,MyNewTool\WObj:=Workobject_1;
        MoveL Target_530,v50,z0,MyNewTool\WObj:=Workobject_1;
        MoveL Target_540,v50,z0,MyNewTool\WObj:=Workobject_1;
        MoveL Target_550,v50,z0,MyNewTool\WObj:=Workobject_1;
        MoveL Target_560,v50,z0,MyNewTool\WObj:=Workobject_1;
        MoveL Target_570,v50,z0,MyNewTool\WObj:=Workobject_1;
        MoveL Target_490_2,v50,z0,MyNewTool\WObj:=Workobject_1;
    ENDPROC
    PROC O()
        MoveL Target_580_2,v50,z0,MyNewTool\WObj:=Workobject_1;
        MoveL Target_580,v50,z0,MyNewTool\WObj:=Workobject_1;
        MoveL Target_590,v50,z0,MyNewTool\WObj:=Workobject_1;
        MoveL Target_600,v50,z0,MyNewTool\WObj:=Workobject_1;
        MoveL Target_610,v50,z0,MyNewTool\WObj:=Workobject_1;
        MoveL Target_620,v50,z0,MyNewTool\WObj:=Workobject_1;
        MoveL Target_630,v50,z0,MyNewTool\WObj:=Workobject_1;
        MoveL Target_640,v50,z0,MyNewTool\WObj:=Workobject_1;
        MoveL Target_650,v50,z0,MyNewTool\WObj:=Workobject_1;
        MoveL Target_660,v50,z0,MyNewTool\WObj:=Workobject_1;
        MoveL Target_670,v50,z0,MyNewTool\WObj:=Workobject_1;
        MoveL Target_680,v50,z0,MyNewTool\WObj:=Workobject_1;
        MoveL Target_690,v50,z0,MyNewTool\WObj:=Workobject_1;
        MoveL Target_700,v50,z0,MyNewTool\WObj:=Workobject_1;
        MoveL Target_710,v50,z0,MyNewTool\WObj:=Workobject_1;
        MoveL Target_720,v50,z0,MyNewTool\WObj:=Workobject_1;
        MoveL Target_730,v50,z0,MyNewTool\WObj:=Workobject_1;
        MoveL Target_740,v50,z0,MyNewTool\WObj:=Workobject_1;
        MoveL Target_580_2,v50,z0,MyNewTool\WObj:=Workobject_1;
        MoveL Target_750_2,v50,z0,MyNewTool\WObj:=Workobject_1;
        MoveL Target_750,v50,z0,MyNewTool\WObj:=Workobject_1;
        MoveL Target_760,v50,z0,MyNewTool\WObj:=Workobject_1;
        MoveL Target_770,v50,z0,MyNewTool\WObj:=Workobject_1;
        MoveL Target_780,v50,z0,MyNewTool\WObj:=Workobject_1;
        MoveL Target_790,v50,z0,MyNewTool\WObj:=Workobject_1;
        MoveL Target_800,v50,z0,MyNewTool\WObj:=Workobject_1;
        MoveL Target_810,v50,z0,MyNewTool\WObj:=Workobject_1;
        MoveL Target_820,v50,z0,MyNewTool\WObj:=Workobject_1;
        MoveL Target_830,v50,z0,MyNewTool\WObj:=Workobject_1;
        MoveL Target_840,v50,z0,MyNewTool\WObj:=Workobject_1;
        MoveL Target_850,v50,z0,MyNewTool\WObj:=Workobject_1;
        MoveL Target_860,v50,z0,MyNewTool\WObj:=Workobject_1;
        MoveL Target_870,v50,z0,MyNewTool\WObj:=Workobject_1;
        MoveL Target_750_2,v50,z0,MyNewTool\WObj:=Workobject_1;
    ENDPROC
    PROC R()
        MoveL Target_880_2,v50,z0,MyNewTool\WObj:=Workobject_1;
        MoveL Target_880,v50,z0,MyNewTool\WObj:=Workobject_1;
        MoveL Target_890,v50,z0,MyNewTool\WObj:=Workobject_1;
        MoveL Target_900,v50,z0,MyNewTool\WObj:=Workobject_1;
        MoveL Target_910,v50,z0,MyNewTool\WObj:=Workobject_1;
        MoveL Target_920,v50,z0,MyNewTool\WObj:=Workobject_1;
        MoveL Target_930,v50,z0,MyNewTool\WObj:=Workobject_1;
        MoveL Target_940,v50,z0,MyNewTool\WObj:=Workobject_1;
        MoveL Target_950,v50,z0,MyNewTool\WObj:=Workobject_1;
        MoveL Target_960,v50,z0,MyNewTool\WObj:=Workobject_1;
        MoveL Target_970,v50,z0,MyNewTool\WObj:=Workobject_1;
        MoveL Target_980,v50,z0,MyNewTool\WObj:=Workobject_1;
        MoveL Target_990,v50,z0,MyNewTool\WObj:=Workobject_1;
        MoveL Target_1000,v50,z0,MyNewTool\WObj:=Workobject_1;
        MoveL Target_1010,v50,z0,MyNewTool\WObj:=Workobject_1;
        MoveL Target_880_2,v50,z0,MyNewTool\WObj:=Workobject_1;
        MoveL Target_1020_2,v50,z0,MyNewTool\WObj:=Workobject_1;
        MoveL Target_1020,v50,z0,MyNewTool\WObj:=Workobject_1;
        MoveL Target_1030,v50,z0,MyNewTool\WObj:=Workobject_1;
        MoveL Target_1040,v50,z0,MyNewTool\WObj:=Workobject_1;
        MoveL Target_1050,v50,z0,MyNewTool\WObj:=Workobject_1;
        MoveL Target_1060,v50,z0,MyNewTool\WObj:=Workobject_1;
        MoveL Target_1070,v50,z0,MyNewTool\WObj:=Workobject_1;
        MoveL Target_1080,v50,z0,MyNewTool\WObj:=Workobject_1;
        MoveL Target_1090,v50,z0,MyNewTool\WObj:=Workobject_1;
        MoveL Target_1100,v50,z0,MyNewTool\WObj:=Workobject_1;
        MoveL Target_1110,v50,z0,MyNewTool\WObj:=Workobject_1;
        MoveL Target_1020_2,v50,z0,MyNewTool\WObj:=Workobject_1;
    ENDPROC
    PROC M()
        MoveL Target_1120_2,v50,z0,MyNewTool\WObj:=Workobject_1;
        MoveL Target_1120,v50,z0,MyNewTool\WObj:=Workobject_1;
        MoveL Target_1130,v50,z0,MyNewTool\WObj:=Workobject_1;
        MoveL Target_1140,v50,z0,MyNewTool\WObj:=Workobject_1;
        MoveL Target_1150,v50,z0,MyNewTool\WObj:=Workobject_1;
        MoveL Target_1160,v50,z0,MyNewTool\WObj:=Workobject_1;
        MoveL Target_1170,v50,z0,MyNewTool\WObj:=Workobject_1;
        MoveL Target_1180,v50,z0,MyNewTool\WObj:=Workobject_1;
        MoveL Target_1190,v50,z0,MyNewTool\WObj:=Workobject_1;
        MoveL Target_1200,v50,z0,MyNewTool\WObj:=Workobject_1;
        MoveL Target_1210,v50,z0,MyNewTool\WObj:=Workobject_1;
        MoveL Target_1220,v50,z0,MyNewTool\WObj:=Workobject_1;
        MoveL Target_1230,v50,z0,MyNewTool\WObj:=Workobject_1;
        MoveL Target_1240,v50,z0,MyNewTool\WObj:=Workobject_1;
        MoveL Target_1250,v50,z0,MyNewTool\WObj:=Workobject_1;
        MoveL Target_1120_2,v50,z0,MyNewTool\WObj:=Workobject_1;
    ENDPROC
    PROC A()
        MoveL Target_1260_2,v50,z0,MyNewTool\WObj:=Workobject_1;
        MoveL Target_1260,v50,z0,MyNewTool\WObj:=Workobject_1;
        MoveL Target_1270,v50,z0,MyNewTool\WObj:=Workobject_1;
        MoveL Target_1280,v50,z0,MyNewTool\WObj:=Workobject_1;
        MoveL Target_1290,v50,z0,MyNewTool\WObj:=Workobject_1;
        MoveL Target_1300,v50,z0,MyNewTool\WObj:=Workobject_1;
        MoveL Target_1310,v50,z0,MyNewTool\WObj:=Workobject_1;
        MoveL Target_1320,v50,z0,MyNewTool\WObj:=Workobject_1;
        MoveL Target_1330,v50,z0,MyNewTool\WObj:=Workobject_1;
        MoveL Target_1340,v50,z0,MyNewTool\WObj:=Workobject_1;
        MoveL Target_1260_2,v50,z0,MyNewTool\WObj:=Workobject_1;
        MoveL Target_1350_2,v50,z0,MyNewTool\WObj:=Workobject_1;
        MoveL Target_1350,v50,z0,MyNewTool\WObj:=Workobject_1;
        MoveL Target_1360,v50,z0,MyNewTool\WObj:=Workobject_1;
        MoveL Target_1370,v50,z0,MyNewTool\WObj:=Workobject_1;
        MoveL Target_1380,v50,z0,MyNewTool\WObj:=Workobject_1;
        MoveL Target_1350_2,v50,z0,MyNewTool\WObj:=Workobject_1;
    ENDPROC
    PROC N()
        MoveL Target_1390_2,v50,z0,MyNewTool\WObj:=Workobject_1;
        MoveL Target_1390,v50,z0,MyNewTool\WObj:=Workobject_1;
        MoveL Target_1400,v50,z0,MyNewTool\WObj:=Workobject_1;
        MoveL Target_1410,v50,z0,MyNewTool\WObj:=Workobject_1;
        MoveL Target_1420,v50,z0,MyNewTool\WObj:=Workobject_1;
        MoveL Target_1430,v50,z0,MyNewTool\WObj:=Workobject_1;
        MoveL Target_1440,v50,z0,MyNewTool\WObj:=Workobject_1;
        MoveL Target_1450,v50,z0,MyNewTool\WObj:=Workobject_1;
        MoveL Target_1460,v50,z0,MyNewTool\WObj:=Workobject_1;
        MoveL Target_1470,v50,z0,MyNewTool\WObj:=Workobject_1;
        MoveL Target_1480,v50,z0,MyNewTool\WObj:=Workobject_1;
        MoveL Target_1490,v50,z0,MyNewTool\WObj:=Workobject_1;
        MoveL Target_1390_2,v50,z0,MyNewTool\WObj:=Workobject_1;
    ENDPROC
    PROC U()
        MoveL Target_1500_2,v50,z0,MyNewTool\WObj:=Workobject_1;
        MoveL Target_1500,v50,z0,MyNewTool\WObj:=Workobject_1;
        MoveL Target_1510,v50,z0,MyNewTool\WObj:=Workobject_1;
        MoveL Target_1520,v50,z0,MyNewTool\WObj:=Workobject_1;
        MoveL Target_1530,v50,z0,MyNewTool\WObj:=Workobject_1;
        MoveL Target_1540,v50,z0,MyNewTool\WObj:=Workobject_1;
        MoveL Target_1550,v50,z0,MyNewTool\WObj:=Workobject_1;
        MoveL Target_1560,v50,z0,MyNewTool\WObj:=Workobject_1;
        MoveL Target_1570,v50,z0,MyNewTool\WObj:=Workobject_1;
        MoveL Target_1580,v50,z0,MyNewTool\WObj:=Workobject_1;
        MoveL Target_1590,v50,z0,MyNewTool\WObj:=Workobject_1;
        MoveL Target_1600,v50,z0,MyNewTool\WObj:=Workobject_1;
        MoveL Target_1610,v50,z0,MyNewTool\WObj:=Workobject_1;
        MoveL Target_1620,v50,z0,MyNewTool\WObj:=Workobject_1;
        MoveL Target_1630,v50,z0,MyNewTool\WObj:=Workobject_1;
        MoveL Target_1640,v50,z0,MyNewTool\WObj:=Workobject_1;
        MoveL Target_1650,v50,z0,MyNewTool\WObj:=Workobject_1;
        MoveL Target_1660,v50,z0,MyNewTool\WObj:=Workobject_1;
        MoveL Target_1670,v50,z0,MyNewTool\WObj:=Workobject_1;
        MoveL Target_1680,v50,z0,MyNewTool\WObj:=Workobject_1;
        MoveL Target_1690,v50,z0,MyNewTool\WObj:=Workobject_1;
        MoveL Target_1700,v50,z0,MyNewTool\WObj:=Workobject_1;
        MoveL Target_1710,v50,z0,MyNewTool\WObj:=Workobject_1;
        MoveL Target_1720,v50,z0,MyNewTool\WObj:=Workobject_1;
        MoveL Target_1500_2,v50,z0,MyNewTool\WObj:=Workobject_1;
    ENDPROC
    PROC E()
        MoveL Target_1730_2,v50,z0,MyNewTool\WObj:=Workobject_1;
        MoveL Target_1730,v50,z0,MyNewTool\WObj:=Workobject_1;
        MoveL Target_1740,v50,z0,MyNewTool\WObj:=Workobject_1;
        MoveL Target_1750,v50,z0,MyNewTool\WObj:=Workobject_1;
        MoveL Target_1760,v50,z0,MyNewTool\WObj:=Workobject_1;
        MoveL Target_1770,v50,z0,MyNewTool\WObj:=Workobject_1;
        MoveL Target_1780,v50,z0,MyNewTool\WObj:=Workobject_1;
        MoveL Target_1790,v50,z0,MyNewTool\WObj:=Workobject_1;
        MoveL Target_1800,v50,z0,MyNewTool\WObj:=Workobject_1;
        MoveL Target_1810,v50,z0,MyNewTool\WObj:=Workobject_1;
        MoveL Target_1820,v50,z0,MyNewTool\WObj:=Workobject_1;
        MoveL Target_1830,v50,z0,MyNewTool\WObj:=Workobject_1;
        MoveL Target_1840,v50,z0,MyNewTool\WObj:=Workobject_1;
        MoveL Target_1850,v50,z0,MyNewTool\WObj:=Workobject_1;
        MoveL Target_1730_2,v50,z0,MyNewTool\WObj:=Workobject_1;
    ENDPROC
    PROC L()
        MoveL Target_1860_2,v50,z0,MyNewTool\WObj:=Workobject_1;
        MoveL Target_1860,v50,z0,MyNewTool\WObj:=Workobject_1;
        MoveL Target_1870,v50,z0,MyNewTool\WObj:=Workobject_1;
        MoveL Target_1880,v50,z0,MyNewTool\WObj:=Workobject_1;
        MoveL Target_1890,v50,z0,MyNewTool\WObj:=Workobject_1;
        MoveL Target_1900,v50,z0,MyNewTool\WObj:=Workobject_1;
        MoveL Target_1910,v50,z0,MyNewTool\WObj:=Workobject_1;
        MoveL Target_1920,v50,z0,MyNewTool\WObj:=Workobject_1;
        MoveL Target_1860_2,v50,z0,MyNewTool\WObj:=Workobject_1;
    ENDPROC
    PROC RAYO()
        MoveL Target_1930_2,v50,z0,MyNewTool\WObj:=Workobject_1;
        MoveL Target_1930,v50,z0,MyNewTool\WObj:=Workobject_1;
        MoveL Target_1940,v50,z0,MyNewTool\WObj:=Workobject_1;
        MoveL Target_1950,v50,z0,MyNewTool\WObj:=Workobject_1;
        MoveL Target_1960,v50,z0,MyNewTool\WObj:=Workobject_1;
        MoveL Target_1970,v50,z0,MyNewTool\WObj:=Workobject_1;
        MoveL Target_1980,v50,z0,MyNewTool\WObj:=Workobject_1;
        MoveL Target_1990,v50,z0,MyNewTool\WObj:=Workobject_1;
        MoveL Target_2000,v50,z0,MyNewTool\WObj:=Workobject_1;
        MoveL Target_2010,v50,z0,MyNewTool\WObj:=Workobject_1;
        MoveL Target_2020,v50,z0,MyNewTool\WObj:=Workobject_1;
        MoveL Target_2030,v50,z0,MyNewTool\WObj:=Workobject_1;
        MoveL Target_2040,v50,z0,MyNewTool\WObj:=Workobject_1;
    ENDPROC

    PROC HOME()
        MoveL Target_2100,v50,z0,MyNewTool\WObj:=Workobject_1;
    ENDPROC
    PROC TC()
        MoveL Target_2160,v50,z0,MyNewTool\WObj:=Workobject_1;
    ENDPROC



ENDMODULE
